// TIA Portal V18 export
TYPE "UDT_AHUsRegulators"
// stored: IsFailsafeCompliant false
   STRUCT
      Cfg : "UDT_AHUsRegulatorsDataType";
      State : "UDT_AHUsRegulatorsDataType";
      Demands { S7_SetPoint := 'True'} : "UDT_AHUsRegDemand";
      FreshAirCoef { S7_SetPoint := 'True'} : "UDT_AHUsFreshAirCoef";
   END_STRUCT;
END_TYPE
